(* IEC 61131-3 sources: axopen.templates/axopen.template.simple/ax/src/templates/starterunit, 5 files *)

(* ---- AutomatSequence.st ---- *)
NAMESPACE axosimple.StarterUnitTemplate
    USING axosimple;
    USING AXOpen.Data;
    USING AXOpen.Core;
    USING System.Strings;

    ///<summary>
    /// Provides automatic mode sequence.
    ///</summary>
    {#ix-set:AttributeName = "<#AUTOMAT#>"}
    {S7.extern=ReadWrite}
    CLASS PUBLIC AutomatSequence
        EXTENDS AXOpen.Core.AxoSequencerContainer IMPLEMENTS IModeContainer
        VAR PUBLIC
            Steps : ARRAY[0..100] OF AxoStep;

            _inspectionResult: BOOL;
            _inspectionValue: LREAL;
            _inspectionData: STRING;

            _comprehensiveResult: AXOpen.Inspectors.AxoComprehensiveResult;
        END_VAR

        VAR PRIVATE
            Objs : REF_TO axosimple.StarterUnitTemplate.UnitObjects;

            _currentId : STRING;

            _dialogAnswer : eDialogAnswer;
            _externalCloseOkSignal : BOOL;
            resutl : IAxoTaskState;
        END_VAR

        METHOD INTERNAL Run
            VAR_INPUT
                inParent : AXOpen.Core.IAxoObject;
                inUnitObjects : REF_TO UnitObjects;
            END_VAR

            IF Objs = NULL THEN
                Objs := inUnitObjects;
            END_IF;

            resutl := Objs^.ProcessData.DataManger.CreateOrUpdate('fasdfa');

            // Result is null!
            resutl.IsDone();

            SUPER.Run(inParent);
        END_METHOD
        ///<summary>
        /// Contains logic of the steps of this sequence
        ///</summary>

        VAR
            _isDone : BOOL;
        END_VAR
        METHOD OVERRIDE Main
            VAR
                forIterator : INT := 0;
                dialogTimeOut : TIME:= t#3000ms;
            END_VAR

            IF (Objs = NULL) THEN
                RETURN;
            END_IF;
            // This sequecner executes the steps in cycles from top to bottom
            // in the same order they are written in the program
            // Each step in the sequence must can be used only once.
            // This sets the sequence to run in cycles (top-botton-top and again).
            THIS.SequenceMode := eAxoSequenceMode#Cyclic;

            IF (Steps[0].Execute(THIS, TRUE, '<#GET ID#>')) THEN
                //-------------------------------------------------------
                Objs^._inspectorDialog.Restore();

                // copy data from setting to station data -> it's a problem with override checks identity
                //ProcessData^ :=  ProcessSettings^;

                Objs^.ProcessData.DataManger.Payload.PartPresence.Data()^.FailTime := TIME#3s;
                Objs^.ProcessData.DataManger.Payload.LoadPosition.Data()^.FailTime := TIME#3s;
                Objs^.ProcessData.DataManger.Payload.JigDataMatrixCode.Data()^.FailTime := TIME#3s;

                Objs^.ProcessData.DataManger.Payload.PartPresence.Data()^.PassTime := TIME#2.5s;
                Objs^.ProcessData.DataManger.Payload.LoadPosition.Data()^.PassTime := TIME#2s;
                Objs^.ProcessData.DataManger.Payload.JigDataMatrixCode.Data()^.PassTime := TIME#2s;

                Objs^.ProcessData.DataManger.Payload.PartPresence.Data()^.RequiredStatus := TRUE;
                Objs^.ProcessData.DataManger.Payload.LoadPosition.Data()^.RequiredMin := 1000.0;
                Objs^.ProcessData.DataManger.Payload.LoadPosition.Data()^.RequiredMax := 2000.0;
                Objs^.ProcessData.DataManger.Payload.JigDataMatrixCode.Data()^.RequiredStatus := 'passCode';

                _currentId := 'newProducedPart';
                THIS.MoveNext();
                //-------------------------------------------------------
            END_IF;

            IF (Steps[1].Execute(THIS, TRUE, '<#GET DATA#>')) THEN
                //-------------------------------------------------------

                resutl := Objs^.ProcessData.DataManger.CreateOrUpdate('fasdfa');
                //resutl.IsDone();
                RETURN;

                IF (Objs^.ProcessData.DataManger.CreateOrUpdate(_currentId).IsDone()) THEN
                    THIS.MoveNext();
                END_IF;
                //-------------------------------------------------------
            END_IF;

            IF (Steps[2].Execute(THIS, TRUE, '<#Dialog notify#>')) THEN
                //-------------------------------------------------------
                _externalCloseOkSignal := CurrentStep.Duration > dialogTimeOut;

                _dialogAnswer := Objs^._dialog.ShowWithExternalClose(THIS, _externalCloseOkSignal)
                .WithOK()
                .WithType(eDialogType#Info)
                .WithCaption('Info caption!')
                .WithText('Info - dialog will be closed by external timeout 2s!').Answer();

                IF( _dialogAnswer = eDialogAnswer#Ok) THEN
                    THIS.MoveNext();
                END_IF;
                //-------------------------------------------------------
            END_IF;

            IF (Steps[3].Execute(THIS, TRUE, '<#Dialog success#>')) THEN
                //-------------------------------------------------------
                _externalCloseOkSignal := CurrentStep.Duration > dialogTimeOut;

                    _dialogAnswer := Objs^._dialog.ShowWithExternalClose(THIS, _externalCloseOkSignal)
                    .WithOK()
                    .WithType(eDialogType#Success)
                    .WithCaption('Success caption!')
                    .WithText('Success - dialog will be closed by external timeout 2s!').Answer();

                    IF( _dialogAnswer = eDialogAnswer#Ok) THEN
                        THIS.MoveNext();
                    END_IF;
                //-------------------------------------------------------
            END_IF;

            IF (Steps[4].Execute(THIS, TRUE, '<#Dialog Warning#>')) THEN
                //-------------------------------------------------------
                _externalCloseOkSignal := CurrentStep.Duration > dialogTimeOut;

                    _dialogAnswer := Objs^._dialog.ShowWithExternalClose(THIS, _externalCloseOkSignal)
                    .WithYesNo()
                    .WithType(eDialogType#Warning)
                    .WithCaption('Warning caption!')
                    .WithText('Warning - dialog will be closed by external timeout 2s!').Answer();

                    IF( _dialogAnswer = eDialogAnswer#Ok) THEN
                        THIS.MoveNext();
                    END_IF;
                //-------------------------------------------------------
            END_IF;

            IF (Steps[5].Execute(THIS, TRUE, '<#Dialog danger#>')) THEN
                //-------------------------------------------------------
                _externalCloseOkSignal := CurrentStep.Duration > dialogTimeOut;

                    _dialogAnswer := Objs^._dialog.ShowWithExternalClose(THIS, _externalCloseOkSignal)
                    .WithYesNoCancel()
                    .WithType(eDialogType#Warning)
                    .WithCaption('Danger caption!')
                    .WithText('Danger - dialog will be closed by external timeout 2s!').Answer();

                    IF( _dialogAnswer = eDialogAnswer#Ok) THEN
                        THIS.MoveNext();
                    END_IF;
                //-------------------------------------------------------
            END_IF;

            IF (Steps[6].Execute(THIS, TRUE, 'Example Digital inspection')) THEN
                //-------------------------------------------------------
                Objs^.ProcessData.DataManger.Payload.PartPresence.WithCoordinator(THIS).Inspect(THIS,_inspectionResult)
                .UpdateComprehensiveResult(_comprehensiveResult)
                .OnFail()
                .CarryOn();
                //-------------------------------------------------------
            END_IF;

            IF (Steps[7].Execute(THIS, TRUE, 'Example Analog inspection')) THEN
                //-------------------------------------------------------
                _inspectionValue := -5500;

                Objs^.ProcessData.DataManger.Payload.LoadPosition.WithCoordinator(THIS)
                .Inspect(THIS,_inspectionValue)
                .UpdateComprehensiveResult(_comprehensiveResult)
                .OnFail()
                .Dialog( inRetryStep := Steps[50], inTerminateStep := Steps[60], inoDialog := Objs^._inspectorDialog);
                //-------------------------------------------------------
            END_IF;

            IF (Steps[8].Execute(THIS, TRUE, 'Example Data inspection')) THEN
                //-------------------------------------------------------
                _inspectionData := 'tempCode';

                Objs^.ProcessData.DataManger.Payload.JigDataMatrixCode.WithCoordinator(THIS)
                .Inspect(THIS,_inspectionData)
                .UpdateComprehensiveResult(_comprehensiveResult)
                .OnFail()
                .Dialog( inRetryStep := Steps[70], inTerminateStep := Steps[80], inoDialog := Objs^._inspectorDialog);
                //-------------------------------------------------------
            END_IF;

            FOR forIterator := 10 TO 89 BY 1 DO
                IF (Steps[forIterator].Execute(THIS, TRUE,Concat('DO SOMETHING -A-',ToString(forIterator)) )) THEN
                    //-------------------------------------------------------
                    IF CurrentStep.Duration > TIME#50ms THEN
                        THIS.MoveNext();
                    END_IF;
                    //-------------------------------------------------------
                END_IF;
            END_FOR;

            IF (Steps[99].Execute(THIS, TRUE,'<#UPDATE DATA#>')) THEN
                //-------------------------------------------------------
                IF (Objs^.ProcessData.DataManger.Update(_currentId).IsDone()) THEN
                    THIS.MoveNext();
                END_IF;
                //-------------------------------------------------------
            END_IF;

            // This will close the sequence and will return to the first step.
            THIS.Close(Steps[100]);
        END_METHOD
    END_CLASS

END_NAMESPACE

(* ---- GroundSequence.st ---- *)
NAMESPACE axosimple.StarterUnitTemplate
    USING axosimple;
    USING AXOpen.Data;
    USING AXOpen.Core;
    USING System.Strings;

    ///<summary>
    /// Provides ground mode sequence.
    ///</summary>
    {#ix-set:AttributeName = "<#GROUND#>"}
    {S7.extern=ReadWrite}
    CLASS PUBLIC GroundSequence
        EXTENDS AXOpen.Core.AxoSequencerContainer IMPLEMENTS IModeContainer
        VAR PUBLIC
            Steps : ARRAY[0..100] OF AXOpen.Core.AxoStep;
            MoveToWork : AXOpen.Core.AxoTask;
        END_VAR
        VAR PRIVATE
            Objs : REF_TO axosimple.StarterUnitTemplate.UnitObjects;
            // Components : REF_TO axosimple.StarterUnitTemplate.Components;
            // ProcessDataManager : REF_TO axosimple.StarterUnitTemplate.ProcessDataManager;
            // ProcessSettingsManager : REF_TO axosimple.StarterUnitTemplate.FragmentProcessDataManger;
            // TechnologySettingsManager : REF_TO axosimple.StarterUnitTemplate.TechnologyDataManager;

            PersistentSettings : REF_TO AxoDataPersistentExchange;

            _currentId : STRING;
            techSetttingsId : STRING;
        END_VAR

        METHOD INTERNAL Run
            VAR_INPUT
                inParent : AXOpen.Core.IAxoObject;
                inUnitObjects : REF_TO axosimple.StarterUnitTemplate.UnitObjects;
            END_VAR

            IF Objs = NULL THEN
                Objs := inUnitObjects;

                // Components := Objs^.Components;
                // ProcessDataManager := Objs^.ProcessData;
                // ProcessSettingsManager := Objs^.ProcessSettings;
                // TechnologySettingsManager := Objs^.TechnologySettings;
                PersistentSettings := Objs^.Global^.PersistentData;
            END_IF;

            SUPER.Run(inParent);
        END_METHOD

        ///<summary>
        /// Contains logic of the steps of this sequence
        ///</summary>
        METHOD PROTECTED OVERRIDE Main
            VAR
                taskState : AXOpen.Core.IAxoTaskState;
                forIterator : INT;
                _dialogAnswer : eDialogAnswer;
            END_VAR;
            // IF (Components = NULL OR ProcessData = NULL) THEN
            //     RETURN;
            // END_IF;
            // This sequecner executes the steps in cycles from top to bottom
            // in the same order they are written in the program
            // Each step in the sequence must can be used only once.
            // This sets the sequence to run once (top-botton) and stops with done after closing.
            THIS.SequenceMode := eAxoSequenceMode#RunOnce;

            IF (Steps[0].Execute(THIS, TRUE, '<#DIALOG#>')) THEN
                //-------------------------------------------------------

                _dialogAnswer := Objs^._dialog.Show(THIS).WithCaption('<#DO YOU WANT TO RUN THE GROUND MODE SEQUENCE?#>').WithYesNo().WithType(eDialogType#Warning).Answer();

                IF(_dialogAnswer <> eDialogAnswer#NoAnswer) THEN
                    IF(_dialogAnswer = eDialogAnswer#Yes) THEN
                        THIS.MoveNext();
                    END_IF;

                    IF(_dialogAnswer = eDialogAnswer#No) THEN
                        THIS.Restore();
                    END_IF;
                END_IF;
                //-------------------------------------------------------
            END_IF;

            // This is more verbose but also more versatile way of executing step logic.
            IF (Steps[1].Execute(THIS, TRUE, '<#RESTORE#>')) THEN
                //-------------------------------------------------------
                IF(Objs <> NULL) THEN
                    Objs^.TechnologySettings^.Restore();
                    Objs^.ProcessData.DataManger.Restore();
                    Objs^._dialog.Restore();
                    Objs^._alertDialog.Restore();
                    Objs^._inspectorDialog.Restore();
                    THIS.MoveNext();
                END_IF;
                //-------------------------------------------------------
            END_IF;

            IF (Steps[2].Execute(THIS, TRUE, '<#READ PERSISTENT SETTINGS#>')) THEN
                //-------------------------------------------------------
                IF CurrentStep.IsFirstEntryToStep() THEN
                    ;// some special initialization
                END_IF;

                CASE TO_INT( THIS.GetMicroStepValue()) OF
                    0 :
                        IF PersistentSettings^.InvokeEntityExist(THIS ,'') THEN
                            THIS.SetMicroStepValue(UINT#10);
                        END_IF;

                    10 :
                        IF PersistentSettings^.IsEntityExistDone(THIS) THEN
                            IF PersistentSettings^.EntityExistResult() THEN
                                THIS.SetMicroStepValue(UINT#40); // default data exist
                            ELSE
                                THIS.SetMicroStepValue(UINT#20); // no data exist
                            END_IF;
                        END_IF;

                    20 :
                        IF PersistentSettings^.InvokeUpdateAll(THIS) THEN // data not exist -> udate all to DB
                            THIS.SetMicroStepValue(UINT#30);
                        END_IF;

                    30:
                        IF PersistentSettings^.IsUpdateAllDone(THIS) THEN
                            THIS.SetMicroStepValue(UINT#40); // all was updated to DB
                        END_IF;

                    40 :
                        IF PersistentSettings^.InvokeRead(THIS, '') THEN // read default group
                            THIS.SetMicroStepValue(UINT#50);
                        END_IF;
                    50 :
                        IF PersistentSettings^.IsReadDone(THIS) THEN
                                THIS.MoveNext(); // just default group was readed
                        END_IF;
                    ELSE
                        THIS.SetMicroStepValue(UINT#0);
                END_CASE;

                //-------------------------------------------------------
            END_IF;

            IF (Steps[5].Execute(THIS, TRUE, '<#READ TECHNOLOGY SETTINS#>')) THEN
                //-------------------------------------------------------

                IF CurrentStep.IsFirstEntryToStep() THEN
                    IF(Objs^.Global = NULL) THEN RETURN; END_IF;
                    IF(Objs^.Global^.TechnologySettings = NULL) THEN RETURN; END_IF;

                    IF Objs^.Global^.TechnologySettings^.Common.Entity.DataEntityId <> '' THEN
                       techSetttingsId := Objs^.Global^.TechnologySettings^.Common.Entity.DataEntityId; // TAKE GLOGAL TECHNOLOGY SETTINGS ID

                    ELSIF Objs^.TechnologySettings^.Payload.DataEntityId <> '' THEN // TAKE LAST LOADED FOR STATION
                        techSetttingsId := Objs^.TechnologySettings^.Payload.DataEntityId;

                    ELSIF Objs^.LastTechnologySettings <> '' THEN // TAKE LAST LOADED FROM PERSISTENT
                        techSetttingsId := Objs^.LastTechnologySettings;
                    ELSE
                        Objs^.LastTechnologySettings := 'default'; // FORCE DEFAULT VALUE
                        techSetttingsId := Objs^.LastTechnologySettings;
                    END_IF;

                    IF Objs^.Global^.TechnologySettings^.Common.Entity.DataEntityId = Objs^.TechnologySettings^.Payload.DataEntityId then
                        //THIS.MoveNext(); // you can skip loading...
                        ;
                    end_if;

                else
                    // IF(Objs^.TechnologySettings^.Read( techSetttingsId ).IsDone()) THEN
                    //     THIS.MoveNext();
                    // END_IF;
                    THIS.MoveNext();
                END_IF;
                //-------------------------------------------------------
            END_IF;

            FOR forIterator := 6 TO 98 BY 1 DO
                IF (Steps[forIterator].Execute(THIS, TRUE,Concat('DO SOMETHING -G-',ToString(forIterator)) )) THEN
                    //-------------------------------------------------------
                    IF CurrentStep.Duration > TIME#25ms THEN
                        THIS.MoveNext();
                    END_IF;
                    //-------------------------------------------------------
                END_IF;
            END_FOR;

            IF (Steps[99].Execute(THIS, TRUE, '<#SAVE DATA#>')) THEN
                //-------------------------------------------------------
                CASE TO_INT( THIS.GetMicroStepValue()) OF
                    0 :
                        IF Objs^.ProcessData.Shared.Entity.DataEntityId <> '' THEN
                            _currentId := Objs^.ProcessData.Shared.Entity.DataEntityId;
                            THIS.SetMicroStepValue(UINT#10);

                        ELSE // FIST RUN OR WITHOUT DATA
                            THIS.MoveNext();
                        END_IF;

                    10 : // update part as a corrupted a interrupted
                        Objs^.ProcessData.Shared.Entity.WasReset := true;
                        IF Objs^.ProcessData.Update(_currentId).IsDone() THEN
                                THIS.MoveNext();
                        END_IF;
                    ELSE
                        THIS.SetMicroStepValue(UINT#0);
                END_CASE;
                //-------------------------------------------------------
            END_IF;

            // This will close the sequence and will return to the first step.
            THIS.Close(Steps[100]);
        END_METHOD
    END_CLASS
END_NAMESPACE

(* ---- ServiceMode.st ---- *)
NAMESPACE axosimple.StarterUnitTemplate
    USING axosimple;
    USING AXOpen.Data;
    USING AXOpen.Core;
    USING System.Strings;

    ///<summary>
    /// Provides logic for service/manual/maintenance mode.
    ///</summary>
    {#ix-set:AttributeName = "<#SERVICE#>"}
    {S7.extern=ReadWrite}
    CLASS PUBLIC ServiceMode
        EXTENDS AXOpen.Core.AxoTask IMPLEMENTS IModeContainer
        ///<summary>
        /// Runs service mode logic. This method must be called cyclically.
        ///</summary>

        METHOD PUBLIC Run
            VAR_INPUT
                parent : IAxoObject;
            END_VAR
            VAR_IN_OUT
                components : axosimple.StarterUnitTemplate.Components;
            END_VAR
            THIS.Initialize(parent);
            IF THIS.Execute() THEN
                THIS.Handle(components);
            END_IF;
        END_METHOD

        METHOD PRIVATE Handle
            VAR_IN_OUT
                components : axosimple.StarterUnitTemplate.Components;
            END_VAR
            ;
            // HERE CALL LOGIC FOR MANUAL/SERICE OPERATIONS
        END_METHOD
    END_CLASS
END_NAMESPACE

(* ---- Unit.st ---- *)
NAMESPACE axosimple.StarterUnitTemplate
    USING axosimple;
    USING AXOpen.Data;
    USING AXOpen.Core;
    USING System.Strings;

    ///<summary>
    /// Represents controlled units and high level task coordination.
    ///</summary>
    {S7.extern=ReadWrite}
    CLASS Unit
        EXTENDS axosimple.BaseUnit.UnitBase
        VAR PUBLIC
            ///<summary>
            /// Provide access to unit objets, that are used into sequnces.
            ///</summary>
            X  : axosimple.StarterUnitTemplate.UnitObjects;

            ///<summary>
            /// Ground sequence. Contains logic that brings the unit into initial state.
            ///</summary>
            Ground : axosimple.StarterUnitTemplate.GroundSequence;

            ///<summary>
            /// Automatic sequence. Contains logic for automatic operations of this unit.
            ///</summary>
            Auto : axosimple.StarterUnitTemplate.AutomatSequence;

            ///<summary>
            /// Service mode contains logic for service/manual operations.
            ///</summary>
            Service : axosimple.StarterUnitTemplate.ServiceMode;
        END_VAR
        ///<summary>
        /// Runs this unit.
        ///</summary>

        METHOD PUBLIC Run
            VAR_INPUT
                inParent : IAxoContext;
            END_VAR
            VAR_IN_OUT
                ///<summary>
                /// Hardware input structure
                ///</summary>
                inoInputs : axosimple.Inputs;
                ///<summary>
                /// Hardware output structure
                ///</summary>
                inoOutputs : axosimple.Outputs;
            END_VAR
            VAR_INPUT
                inGlobal : REF_TO axosimple.GlobalContextObjects;
            END_VAR
            THIS.Initialize(inParent);
            X.G := inGlobal;
            THIS.Execute(inoInputs, inoOutputs);
        END_METHOD

        ///<summary>
        ///     Exectute for this unit.
        ///     Execute runs cyclicaly you should place any call of this unit in this or underlying methods.
        ///</summary>
        METHOD PRIVATE Execute
            VAR_IN_OUT
                inoInputs : axosimple.Inputs;
                inoOutputs : axosimple.Outputs;
            END_VAR

            // Component I/O immange and management handling.
             X.C.Update(THIS, inoInputs, inoOutputs);

             // Run process data manager of this unit.
             X.PD.Run(THIS);

             // Run technology data manger of this unit.
             X.TD.Run(THIS);

            /*

                    Ground mode handling

            */

             Ground.Run(THIS, REF(X));

             // Restores other states when Ground executes
             IF (Ground.IsBusy()) THEN
                 Auto.Restore();
                 Service.Restore();
             END_IF;

             /*

                    Automatic mode handling
                    NOTE: Ground must be previously done.

             */

             Auto.IsDisabled := Ground.Status <> eAxoTaskState#Done;
             Auto.Run(THIS, REF(X));

            /*

                Service/manual mode hadnling

             */

             Service.Run(THIS, X.C);

             IF Service.IsBusy() THEN
                 Ground.Restore();
                 Auto.Restore();
             END_IF;

        END_METHOD
    END_CLASS
END_NAMESPACE

(* ---- UnitObjects.st ---- *)
NAMESPACE axosimple.StarterUnitTemplate

    USING axosimple;
    USING AXOpen.Data;
    USING AXOpen.Core;
    USING System.Strings;

    {S7.extern=ReadWrite}
    CLASS PUBLIC UnitObjects EXTENDS axosimple.BaseUnit.UnitObjects
        VAR PUBLIC
            ///<summary>
            /// Handles and intializes components used by this unit.
            ///</summary>
            Components : axosimple.StarterUnitTemplate.Components;

            ///<summary>
            /// Provides access to process data manager of this unit.
            ///</summary>
            ProcessData : axosimple.StarterUnitTemplate.ProcessDataManager;

            ///<summary>
            /// Provides access to technology data managers of this unit.
            ///</summary>
            TechnologyData : axosimple.StarterUnitTemplate.TechnologyDataManager;

            ///<summary>
            /// Provides access to process data manager of this unit.
            ///</summary>
            TechnologySettings : REF_TO axosimple.StarterUnitTemplate.FragmentTechnologyDataManger;

            ///<summary>
            /// Provides access to process data manager of this unit.
            ///</summary>
            ProcessSettings : REF_TO axosimple.StarterUnitTemplate.FragmentProcessDataManger;

            {#ix-attr:[AXOpen.Data.PersistentAttribute("StarterUnitTemplate")]}
            SpecialSettings :STRING[64] ;

            // https://ix-ax.github.io/AXOpen/core/docs/AXODIALOG.html#closing-a-dialog-with-external-signal
            _dialog : AXOpen.Core.AxoDialog;

            // https://ix-ax.github.io/AXOpen/core/docs/AXOALERTDIALOG.html#invoking-alerts-from-plc
            _alertDialog : AXOpen.Core.AxoAlert;

            // it needs to be handle from auto or ground sequnce
            _inspectorDialog       : AXOpen.Inspectors.AxoInspectorDialog;

        END_VAR
    END_CLASS

END_NAMESPACE
